FUNCTION_BLOCK M_commands_handling
VAR_INPUT
	CommandNumberl:UINT;
END_VAR
VAR_OUTPUT
END_VAR
VAR
END_VAR

END_FUNCTION_BLOCK

(* stored: Version 1.1.0.1, ProductVersion 3.1.4024.9
   POU M_commands_handling: Id {f452c0c4-a3e8-424a-b858-948b3c779d51}, SpecialFunc None *)
